TYPE ST_AxisPosPar :
STRUCT
	bRelEnable			:BOOL		;		//FALSE绝对定位，TRUE相对定位	
	rPos				:REAL		;		//定位位置	
	rVel				:REAL		;		//定位速度	
	rAcc				:REAL		;		//定位加速度	
	rDec				:REAL		;		//定位减速度	
	rJerk				:REAL		;		//定位跃度	
END_STRUCT
END_TYPE

(* stored: Version 1.1.0.1, ProductVersion 3.1.4024.12
   DUT ST_AxisPosPar: Id {cf6f22f8-8818-4674-b683-bb2d26741a41} *)
